(*

.. <legal notes>

legal notes
=================
| SPDX-FileCopyrightText: © 2026 Oleksandr Tiutyk <trofimich@gmail.com>
| SPDX-License-Identifier: LGPL-3.0-only
| For details check: LGPL-3.0-only_

.. _LGPL-3.0-only: https://www.gnu.org/licenses/lgpl-3.0.en.html

.. </legal notes>

*)

PROGRAM LongRealHelper
VAR CONSTANT
	MIN_VALUE : LREAL := -1.7976931348623158E+308;
	MAX_VALUE : LREAL := +1.7976931348623158E+308;
END_VAR
VAR
	_ClassName : STRING := __POUNAME();
END_VAR

{attribute 'monitoring' := 'call'}
PROPERTY ClassName : STRING
GET
ClassName := _ClassName;
END_GET
END_PROPERTY

{attribute 'monitoring' := 'call'}
PROPERTY NamespaceName : STRING
GET
NamespaceName := CurrentNamespace.Name;
END_GET
END_PROPERTY

END_PROGRAM

(* stored: Version 1.1.0.1
   POU LongRealHelper: Id {8e3c2d57-ec4d-4c6a-97da-06811177b941}, SpecialFunc None
   Property ClassName: Id {dec151f8-ad14-4f84-8a65-a10b7a729f04}
   Get Get: Id {609b9324-4979-4f22-9ee4-d3b56f82666c}
   Property NamespaceName: Id {3472afc4-85a8-4119-a5ca-dd94ad244223}
   Get Get: Id {bb7fe1cc-c438-48fc-b6cd-d6a3e2da25f3} *)
